TYPE ST_ORCA_Outers :
STRUCT
	Code 	: STRING(255);
	xPos		: INT;
	yPos		: INT;

END_STRUCT
END_TYPE

(* stored: Version 1.1.0.1
   DUT ST_ORCA_Outers: Id {7203581f-5f54-43a2-8e5d-a09454fd6aa2} *)
